// TIA Portal project "PID_ControlHeat" (V19)

(* hardware
DEVICE "S7-1500/ET200MP station_1"  S7-1500 station
   slot 0: "Rail_0"  Rack  6ES7 590-1***0-0AA0
   slot 1: "PLC_1"  CPU 1511-1 PN  6ES7 511-1AK02-0AB0  V2.9
      slot 3: "CPU display_1"  6ES7591-1AA00-0AA0
      slot 32768: "PROFINET interface_1"  X1
         slot 32769: "Port_1"  X1 P1
         slot 32770: "Port_2"  X1 P2
      slot 34817: "Virtual CP interface port_1"  Virtual CP interface port  Virtual CP interface port
*)

// ===== PLC "PLC_1"  CPU 1511-1 PN =====

DATA_BLOCK "Pars"   // DB1
{ S7_Optimized_Access := 'TRUE' }
VERSION : 0.1
   VAR
      Temp_SP : Real;
      Temp_PV : Real;
      Power : Real;
      Kp : Real := -1.7;
      Ti : Time := T#78s;
      COM_RST : Bool;
      MAN_ON : Bool;
   END_VAR
BEGIN
END_DATA_BLOCK

DATA_BLOCK "Model_DB"   // DB2
{ S7_Optimized_Access := 'TRUE' }
VERSION : 0.1
// stored: InstanceOfName Model
"Model"
BEGIN
END_DATA_BLOCK

FUNCTION_BLOCK "Model"   // FB1, SCL
{ S7_Optimized_Access := 'TRUE' }
VERSION : 0.1
   VAR_INPUT
      CO : Real := 39.0;
   END_VAR
   VAR_OUTPUT
      PV : Real := 140.0;
   END_VAR
   VAR
      CO_Delay : Array[1..48] of Real;
      PV1 : Real := 140.0;
      Index : Int := 1;
   END_VAR
BEGIN
   IF #Index <= 48 THEN
       #CO_Delay[#Index] := #CO;
   ELSE
       #PV := 0.987 * #PV1 - 0.006929 * #CO_Delay[#Index - 48] + 2.048;
       #PV1 := #PV;
       #CO_Delay[#Index - 48] := #CO;
       IF ((#Index-48) >= 48) THEN
           #Index := 48;
       END_IF;
   END_IF;
   #Index := #Index + 1;
END_FUNCTION_BLOCK

ORGANIZATION_BLOCK "Main"   // OB1, LAD, ProgramCycle
TITLE = "Main Program Sweep (Cycle)"
{ S7_Optimized_Access := 'TRUE' }
VERSION : 0.1
   VAR_INPUT
      Initial_Call : Bool;   // Initial call of this OB
      Remanence : Bool;   // =True, if remanent data are available
   END_VAR
BEGIN
END_ORGANIZATION_BLOCK

ORGANIZATION_BLOCK "CyclicInterrupt"   // OB30, FBD, CyclicInterrupt
{ S7_Optimized_Access := 'TRUE' }
VERSION : 0.1
   VAR_INPUT
      Initial_Call : Bool;   // Initial call of this OB
      Event_Count : Int;   // Events discarded
   END_VAR
BEGIN

REGION Network 1
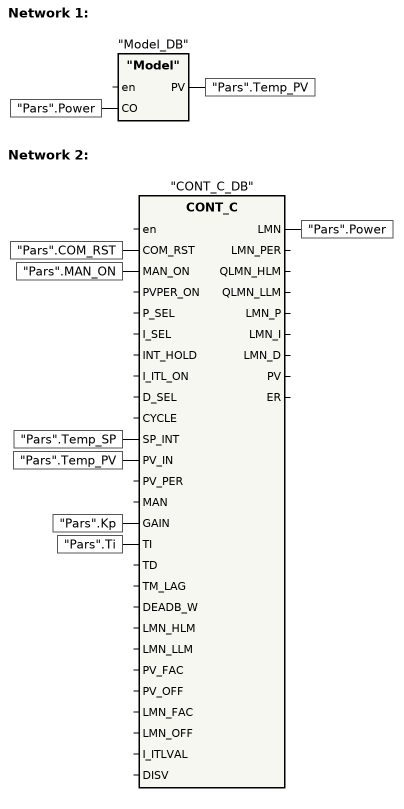
   "Model_DB"(CO := "Pars".Power, PV => "Pars".Temp_PV);   // "Model"
END_REGION

REGION Network 2
   "CONT_C_DB"(COM_RST := "Pars".COM_RST,   // CONT_C
               MAN_ON := "Pars".MAN_ON,
               SP_INT := "Pars".Temp_SP,
               PV_IN := "Pars".Temp_PV,
               GAIN := "Pars".Kp,
               TI := "Pars".Ti,
               LMN => "Pars".Power);
END_REGION
END_ORGANIZATION_BLOCK